(* CODESYS project TrafficLight_completo.project

Project tree, tasks and I/O mapping:
  Device : CODESYS Control Win V3, 3S - Smart Software Solutions GmbH, order no. 305021, version 3.5.10.30
    application Application
      libraries: Standard, * (System)
      task MainTask (cyclic, interval t#20ms, priority 1) calls PLC_PRG
      task VISU_TASK (cyclic, interval 100 ms, priority 31) calls VisuElems.Visu_Prg
      program PLC_PRG [FBD]
      function block NormalCycle [ST]
      visualisation Visualization
  text list GlobalTextList
*)

// Device/Application/PLC_PRG
PROGRAM PLC_PRG
VAR
	Contact1: BOOL; 	
	Contact2: BOOL;
	Contactp: BOOL;
	Contactblink: BOOL;
	coil1: BOOL;
	coil2: BOOL;
	coil3: BOOL; 
	FB:NormalCycle;
	
	TON: TON;
	ET: TIME;
END_VAR

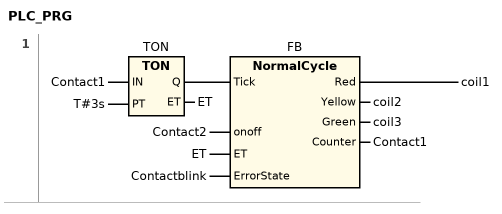
// NETWORK 1
TON(IN := Contact1, PT := T#3s, ET => ET);
FB(
    Tick := TON.Q,
    onoff := Contact2,
    ET := ET,
    ErrorState := Contactblink,
    Yellow => coil2,
    Green => coil3,
    Counter => Contact1); // NormalCycle
coil1 := FB.Red;

END_PROGRAM

// Device/Application/NormalCycle
FUNCTION_BLOCK NormalCycle
VAR_INPUT
	Tick: BOOL;
	onoff: BOOL := FALSE;  
	ET: TIME;
	ErrorState:BOOL;
END_VAR
VAR_OUTPUT
	Red : BOOL:=FALSE;
	Yellow : BOOL:=FALSE;
	Green : BOOL:=FALSE;
	Counter : BOOL;
END_VAR
VAR
	status : INT := 0;
	NextState: INT:=1;
END_VAR

IF onoff = TRUE THEN
	IF ErrorState=TRUE THEN
		status:=4;
	END_IF
		Counter:=TRUE;
		IF Tick THEN 
			status := NextState;
			Counter := FALSE;
			
		END_IF
		CASE status OF 
		0:green := FALSE; red := FALSE; yellow:= FALSE;
		1:green := FALSE; red := TRUE; yellow:= FALSE; NextState:=2; 
		2:green := TRUE; red := FALSE; yellow:= FALSE; NextState:=3; 
		3:green := FALSE; red := FALSE; yellow:= TRUE; NextState:=1; 
		4:green := TRUE; red := TRUE; yellow:= TRUE;	
		END_CASE

ELSE
	green := FALSE; red := FALSE; yellow:= FALSE;
	status:=0;
	Counter := FALSE;
	NextState:=1;
END_IF

END_FUNCTION_BLOCK

// Device/Application/Visualization
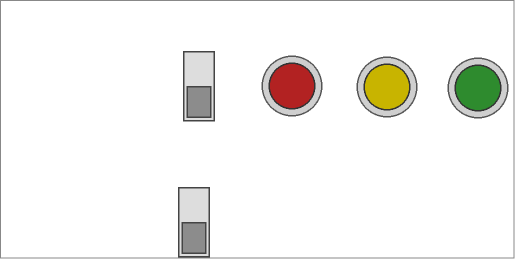
VISUALIZATION Visualization  // 515x259
    Lamp1 (257,51 70x70), variable: PLC_PRG.coil1, style: Lamp-Lamp1-Red
    Lamp1 (352,52 70x70), variable: PLC_PRG.coil2, style: Lamp-Lamp1-Yellow
    Lamp1 (443,53 70x70), variable: PLC_PRG.coil3, style: Lamp-Lamp1-Green
    DipSwitch (164,51 70x70), variable: PLC_PRG.Contact2, behaviour: TOGGLE, style: Switch-DipSwitch-Gray
    DipSwitch (159,187 70x70), tooltip "ERRORSTATE", variable: PLC_PRG.Contactblink, behaviour: TOGGLE, style: Switch-DipSwitch-Gray
END_VISUALIZATION
